// TIA Portal V19 export
ORGANIZATION_BLOCK "A02_OB1"   // OB126, LAD, ProgramCycle
TITLE = "Main Program Sweep (Cycle)"
// stored: SetENOAutomatically false
   VAR_INPUT
      Initial_Call : Bool;   // Initial call of this OB
      Remanence : Bool;   // =True, if remanent data are available
   END_VAR
BEGIN

REGION Network 1: 588 - CU320
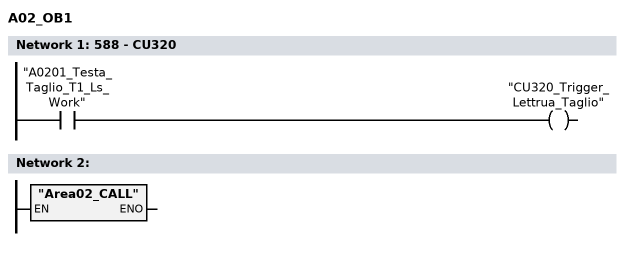
   RUNG wire#powerrail
      Contact( "A0201_Testa_Taglio_T1_Ls_Work" )
      Coil( "CU320_Trigger_Lettrua_Taglio" )
   END_RUNG
   // the same network as SCL:
   "CU320_Trigger_Lettrua_Taglio" := "A0201_Testa_Taglio_T1_Ls_Work";
END_REGION

REGION Network 2
   RUNG wire#powerrail
      "Area02_CALL"()
   END_RUNG
   // the same network as SCL:
   "Area02_CALL"();
END_REGION
END_ORGANIZATION_BLOCK
